FUNCTION_BLOCK B_DEMUX_BOOL (* Basic Function Block Type *)
  (* Standard: 61499-2 *)
  (* Version 0.0, 2015-11-12, 4DIAC-IDE, 4DIAC-Consortium *)
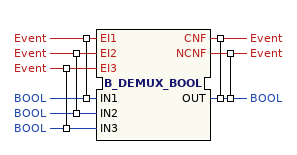
  EVENT_INPUT
    EI1 WITH IN1;
    EI2 WITH IN2;
    EI3 WITH IN3;
  END_EVENT
  EVENT_OUTPUT
    CNF WITH OUT;
    NCNF WITH OUT;
  END_EVENT
  VAR_INPUT
    IN1 : BOOL;
    IN2 : BOOL;
    IN3 : BOOL;
  END_VAR
  VAR_OUTPUT
    OUT : BOOL;
  END_VAR
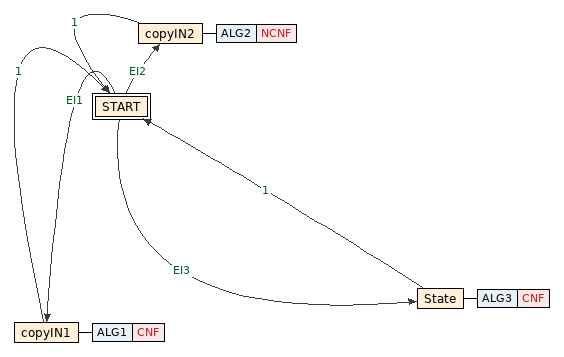
  EC_STATES
    START; (* Initial State *)
    copyIN2 : ALG2 -> NCNF; (* Initialization *)
    copyIN1 : ALG1 -> CNF; (* Normal execution *)
    State : ALG3 -> CNF;
  END_STATES
  EC_TRANSITIONS
    START TO copyIN2 := EI2;
    copyIN2 TO START := 1;
    START TO copyIN1 := EI1;
    copyIN1 TO START := 1;
    START TO State := EI3;
    State TO START := 1;
  END_TRANSITIONS
  ALGORITHM ALG1 IN ST: (* new algorithm *)
OUT:=IN1;
  END_ALGORITHM
  ALGORITHM ALG2 IN ST: (* new algorithm *)
OUT:=IN2;
  END_ALGORITHM
  ALGORITHM ALG3 IN ST: (* new algorithm *)
OUT:=IN3;
  END_ALGORITHM
END_FUNCTION_BLOCK
